{attribute 'qualified_only'}
VAR_GLOBAL
    // Arbiter linked to the FFO and the MPS
    {attribute 'pytmc' := 'pv: PLC:DREAM:MOTION:ARB:01'}
    fbArbiter: FB_Arbiter(1);

    {attribute 'pytmc' := 'pv: PLC:DREAM:MOTION:FFO:02'}
    {attribute 'TcLinkTo' := '.q_xFastFaultOut:=TIIB[PMPS_FFO]^Channel 2^Output'}
    fbFastFaultOutput1: FB_HardwareFFOutput := (bAutoReset := TRUE, i_sNetID:='172.21.92.73.1.1');
END_VAR

(* stored: Version 1.1.0.1
   GVL GVL_PMPS: Id {49a7e34f-b707-4be1-80aa-fd3d166495e3} *)
